// TIA Portal V17 export
// export: Created 2023-02-25T15:47:10.7174905Z, ExportSetting WithDefaults, DisplayName Totally Integrated Automation Portal, DisplayVersion V17, DisplayName TIA Portal Openness, DisplayVersion V17, DisplayName TIA Portal Version Control Interface, DisplayVersion V17, DisplayName TIA Portal Test Suite Advanced, DisplayVersion V17, DisplayName STEP 7 Professional, DisplayVersion V17, DisplayName SIMATIC Energy Suite, DisplayVersion V17, DisplayName STEP 7 Safety, DisplayVersion V17, DisplayName WinCC Professional, DisplayVersion V17
FUNCTION "LOG_AssignmentIOMode" : Void   // FC26, LAD
{ S7_Optimized_Access := 'TRUE' }
VERSION : 0.1
// stored: AutoNumber true, IsIECCheckEnabled false, SetENOAutomatically false, UDAEnableTagReadback false
   VAR_INPUT
      ConveyorsAuto : "stt_Conveyor";
      ConveyorsManual : "stt_Conveyor";
   END_VAR
   VAR_OUTPUT
      C1 : "stt_Motor";
      C2 : "stt_Motor";
      C3 : "stt_Motor";
      C4 : "stt_Motor";
      W : Bool;
      SendLeft : Bool;
      SendForward : Bool;
      SendRight : Bool;
   END_VAR
BEGIN

REGION Network 1: C1
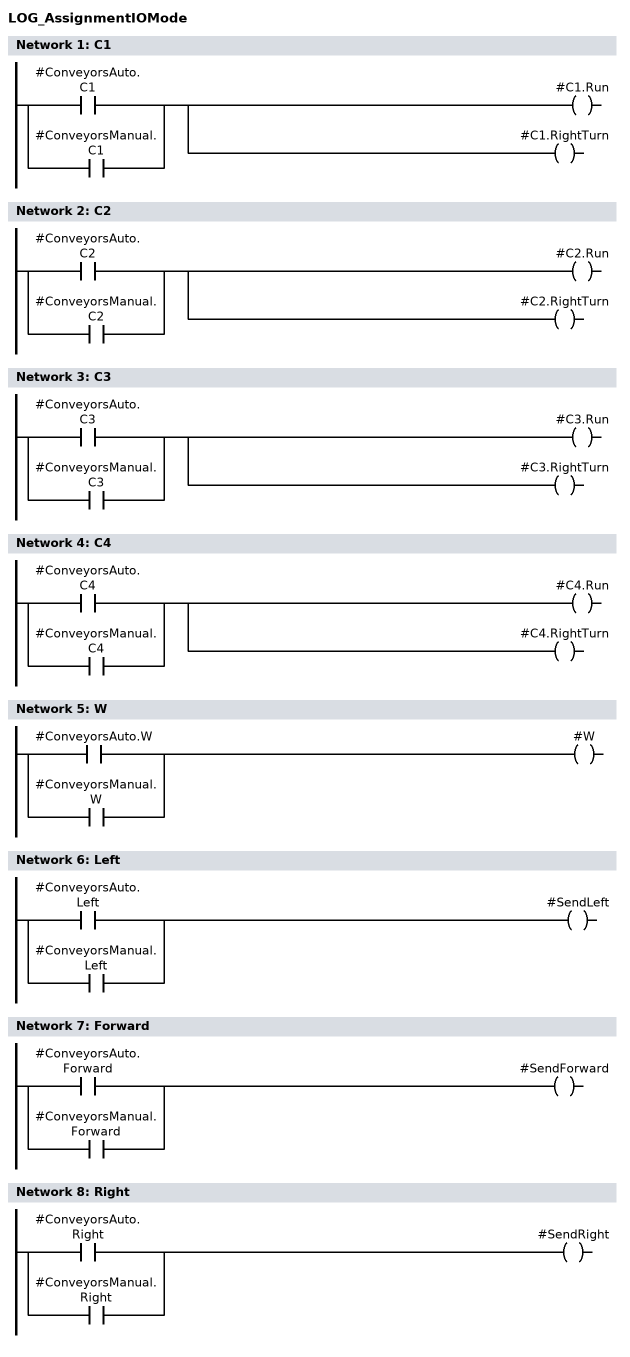
   RUNG wire#powerrail
      Contact( #ConveyorsAuto.C1 )
      wire#w1
      Coil( #C1.Run )
   END_RUNG
   RUNG wire#powerrail
      Contact( #ConveyorsManual.C1 )
   END_RUNG wire#w1
   RUNG wire#w1
      Coil( #C1.RightTurn )
   END_RUNG
   // the same network as SCL:
   #C1.Run := #ConveyorsAuto.C1 OR #ConveyorsManual.C1;
   #C1.RightTurn := #C1.Run;
END_REGION

REGION Network 2: C2
   RUNG wire#powerrail
      Contact( #ConveyorsAuto.C2 )
      wire#w1
      Coil( #C2.Run )
   END_RUNG
   RUNG wire#powerrail
      Contact( #ConveyorsManual.C2 )
   END_RUNG wire#w1
   RUNG wire#w1
      Coil( #C2.RightTurn )
   END_RUNG
   // the same network as SCL:
   #C2.Run := #ConveyorsAuto.C2 OR #ConveyorsManual.C2;
   #C2.RightTurn := #C2.Run;
END_REGION

REGION Network 3: C3
   RUNG wire#powerrail
      Contact( #ConveyorsAuto.C3 )
      wire#w1
      Coil( #C3.Run )
   END_RUNG
   RUNG wire#powerrail
      Contact( #ConveyorsManual.C3 )
   END_RUNG wire#w1
   RUNG wire#w1
      Coil( #C3.RightTurn )
   END_RUNG
   // the same network as SCL:
   #C3.Run := #ConveyorsAuto.C3 OR #ConveyorsManual.C3;
   #C3.RightTurn := #C3.Run;
END_REGION

REGION Network 4: C4
   RUNG wire#powerrail
      Contact( #ConveyorsAuto.C4 )
      wire#w1
      Coil( #C4.Run )
   END_RUNG
   RUNG wire#powerrail
      Contact( #ConveyorsManual.C4 )
   END_RUNG wire#w1
   RUNG wire#w1
      Coil( #C4.RightTurn )
   END_RUNG
   // the same network as SCL:
   #C4.Run := #ConveyorsAuto.C4 OR #ConveyorsManual.C4;
   #C4.RightTurn := #C4.Run;
END_REGION

REGION Network 5: W
   RUNG wire#powerrail
      Contact( #ConveyorsAuto.W )
      wire#w1
      Coil( #W )
   END_RUNG
   RUNG wire#powerrail
      Contact( #ConveyorsManual.W )
   END_RUNG wire#w1
   // the same network as SCL:
   #W := #ConveyorsAuto.W OR #ConveyorsManual.W;
END_REGION

REGION Network 6: Left
   RUNG wire#powerrail
      Contact( #ConveyorsAuto.Left )
      wire#w1
      Coil( #SendLeft )
   END_RUNG
   RUNG wire#powerrail
      Contact( #ConveyorsManual.Left )
   END_RUNG wire#w1
   // the same network as SCL:
   #SendLeft := #ConveyorsAuto.Left OR #ConveyorsManual.Left;
END_REGION

REGION Network 7: Forward
   RUNG wire#powerrail
      Contact( #ConveyorsAuto.Forward )
      wire#w1
      Coil( #SendForward )
   END_RUNG
   RUNG wire#powerrail
      Contact( #ConveyorsManual.Forward )
   END_RUNG wire#w1
   // the same network as SCL:
   #SendForward := #ConveyorsAuto.Forward OR #ConveyorsManual.Forward;
END_REGION

REGION Network 8: Right
   RUNG wire#powerrail
      Contact( #ConveyorsAuto.Right )
      wire#w1
      Coil( #SendRight )
   END_RUNG
   RUNG wire#powerrail
      Contact( #ConveyorsManual.Right )
   END_RUNG wire#w1
   // the same network as SCL:
   #SendRight := #ConveyorsAuto.Right OR #ConveyorsManual.Right;
END_REGION
END_FUNCTION
